INTERFACE I_Skill

METHOD M_Reset : BOOL
VAR_INPUT
END_VAR
END_METHOD

METHOD M_Start : BOOL
VAR_INPUT
END_VAR
END_METHOD

METHOD M_Stop : BOOL
VAR_INPUT
END_VAR
END_METHOD

PROPERTY P_State : eSkillState
GET
END_GET
END_PROPERTY

END_INTERFACE

(* stored: Version 1.1.0.1
   Itf I_Skill: Id {79365a28-22d5-4055-8e0f-322026c09656}
   Method M_Reset: Id {227d86f9-4e42-4255-a6a7-0cb1ef12d3bf}
   Method M_Start: Id {1f05b972-1a8e-40a6-bc9b-2e5c262cfe45}
   Method M_Stop: Id {162fe344-3e11-4662-868f-a597c3443d6e}
   Property P_State: Id {40e7dda2-282e-4f7c-8006-bae5f0f4bd33}
   Get Get: Id {2507897d-5d2e-4ba8-b5fd-d6a23c7d43fb} *)
